INTERFACE IClock

PROPERTY DateTimeInitialised : BOOL
GET
END_GET
END_PROPERTY

PROPERTY NowAsDateTime : DT
GET
END_GET
END_PROPERTY

PROPERTY NowAsTimeStruct : REFERENCE TO TIMESTRUCT
GET
END_GET
END_PROPERTY

END_INTERFACE

(* stored: Version 1.1.0.1, ProductVersion 3.1.4024.3
   Itf IClock: Id {e9193702-7ff6-40fe-8066-15d736a886cb}
   Property DateTimeInitialised: Id {7a53f007-62a7-4176-a25f-0a370f84481b}
   Get Get: Id {3fbf7ef8-f3a8-46a8-9f7c-5852cde6f7d8}
   Property NowAsDateTime: Id {e8a117e8-04ae-46c5-b979-9a96cfcad643}
   Get Get: Id {78d8418f-f664-43c8-b3bb-52188ae91793}
   Property NowAsTimeStruct: Id {95e89d62-9c91-4a9d-9163-c909693c369b}
   Get Get: Id {5b539b93-9af1-4697-8cb5-23b865126c16} *)
